(* Logix 5000 project; controller AplicacionAFEbancoDePruebas vendor 1 type 14 code 149 rev 33.12; software revision 33.01 *)

TASK MainTask (continuous, watchdog 500 ms) : MainProgram

MODULES
   Local : vendor 1 type 14 code 149 (Compact 0, rev 33.12)
      Discrete_IO : Embedded (Compact 1, rev 3.1, Output RPI 20 ms)
      PLC : 1769-L32E Ethernet Port (Ethernet 192.168.2.131, rev 20.1)
         PLC_Controller : vendor 1 type 14 code 77 (CompactLogixL32EController 0, rev 20.1, $23548359$ RPI 20 ms)
      VSD_AFE : vendor 1 type 143 code 8336 (Ethernet 192.168.2.50, rev 6.5, Output RPI 20 ms)
          : vendor 1 type 143 code 416 (RhinoBP 4, rev 1.8)
          : vendor 1 type 143 code 416 (RhinoBP 5, rev 1.8)
          : vendor 1 type 143 code 161 (RhinoBP 10, rev 1.1)
          : vendor 1 type 143 code 4770 (RhinoBP 12, rev 1.1)
          : vendor 1 type 143 code 675 (RhinoBP 13, rev 1.1)
          : vendor 1 type 143 code 2724 (RhinoBP 14, rev 1.1)
END_MODULES

TYPE Dinagrama :   // Estructura para el dinagrama
STRUCT
   vPotencia : REAL[500];
   NumeroMuestras : INT;
END_STRUCT
END_TYPE

TYPE SWC :
STRUCT
   Dinagrama : Dinagrama;
END_STRUCT
END_TYPE

VAR_GLOBAL   (* controller tags *)
   SRP_SimActualStroke : DINT;   // Variable Simulación de PLC Variador DC
   SWC : SWC;
   TestValueFlag : BOOL;
END_VAR

PROGRAM MainProgram   (* main routine MainRoutine *)
VAR
   Captura : BOOL;
   contadorAux : ALIAS FOR counter[0].ACC;
   counter : COUNTER[10];
   Enabled : BOOL;
   Flag : BOOL;
   habilitar : DINT;
   myoneshot : BOOL[32];
        [0]   // oneshot toogle bot dinagrama
   Proximetro_Virtual : ALIAS FOR SRP_SimActualStroke;
   SPM_Reference : REAL;
   timer : TIMER[10] := ([0].PRE := 2000, [0].ACC := 895, [0].EN := 1, [0].TT := 1);
        [0]   // Tiempo Muestreo
END_VAR

ROUTINE dinagramaPotencia   (* ladder *)
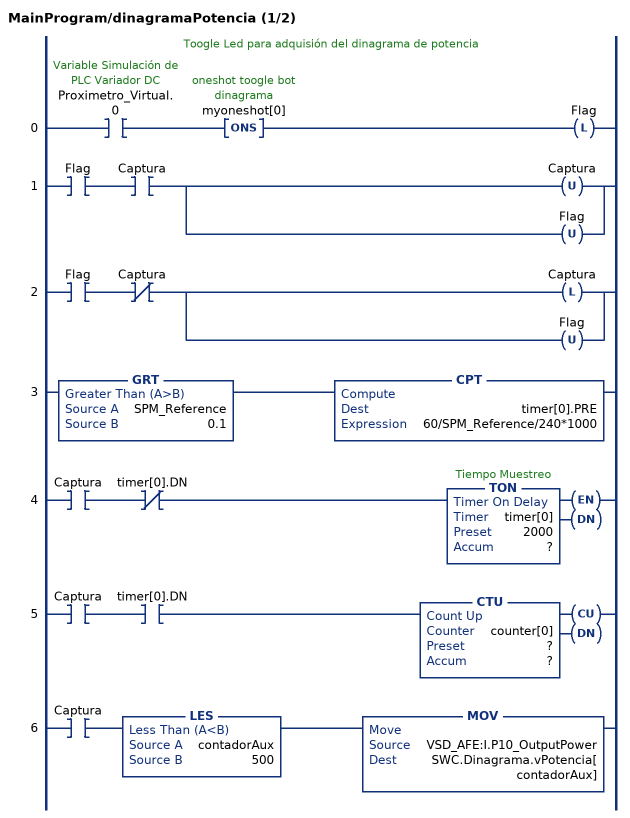
   // Toogle Led para adquisión del dinagrama de potencia
   0: XIC(Proximetro_Virtual.0)ONS(myoneshot[0])OTL(Flag);
   1: XIC(Flag)XIC(Captura)[OTU(Captura) ,OTU(Flag) ];
   2: XIC(Flag)XIO(Captura)[OTL(Captura) ,OTU(Flag) ];
   3: GRT(SPM_Reference,0.1)CPT(timer[0].PRE,60/SPM_Reference/240*1000);
   4: XIC(Captura)XIO(timer[0].DN)TON(timer[0],?,?);
   5: XIC(Captura)XIC(timer[0].DN)CTU(counter[0],?,?);
   6: XIC(Captura)LES(contadorAux,500)MOV(VSD_AFE:I.P10_OutputPower,SWC.Dinagrama.vPotencia[contadorAux]);
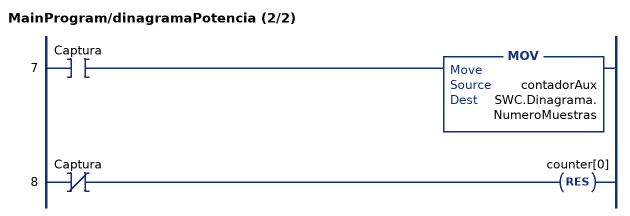
   7: XIC(Captura)MOV(contadorAux,SWC.Dinagrama.NumeroMuestras);
   8: XIO(Captura)RES(counter[0]);
END_ROUTINE

ROUTINE MainRoutine   (* ladder *)
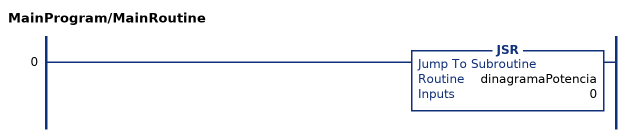
   0: JSR(dinagramaPotencia,0);
END_ROUTINE
END_PROGRAM
